// TIA Portal V18 export
TYPE "UDT_StaProcessData"
   STRUCT
      TypeName : String[50];   // 产品类型
      PartID : String[48];   // 产品序列号
      PalletNo : Int;   // 托盘号
      Mode : Int;   // 作业模式
      "P-SubPartID" : Array[1..10] of String[48];   // 子零件号
      Count_Total : DInt;   // 加工总数
      Count_OK : DInt;   // 合格计数
      Count_NG : DInt;   // 不合格计数
      CycleTime : Real;   // 循环时间
      PartResult : Int;   // 0-未作，1-合格，2-不合格
   END_STRUCT;
END_TYPE
